PROGRAM analogSignals_ex01_1
VAR
	Frawsensor		: REAL;
	fScaledvalue	: real;
	
	LIN_TRAFO 		: FB_Scale;
END_VAR

LIN_TRAFO(
	fIN:= frawsensor, 
	fIN_min:= 4, 
	fIN_max:= 20, 
	fOUT_min:= 0, 
	fOUT_max:= 100, 
	fOUT=> fScaledvalue);

END_PROGRAM

(* stored: Version 1.1.0.1
   POU analogSignals_ex01_1: Id {67f6ed86-298f-49bf-b720-b209da7f3dd0}, SpecialFunc None *)
